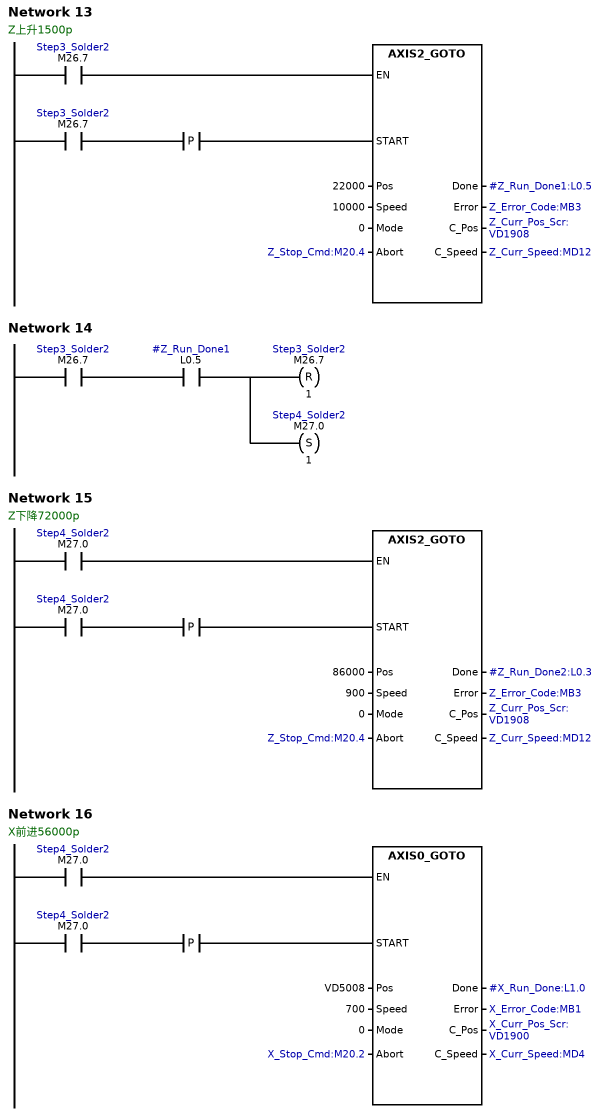
[picture p48: SBR39 networks 13-16]
Network 13
// Z上升1500p
LD     Step3_Solder2:M26.7
=      L60.0
LD     Step3_Solder2:M26.7
EU
=      L63.7
LD     L60.0
CALL   AXIS2_GOTO:SBR25, L63.7, 22000, 10000, 0, Z_Stop_Cmd:M20.4, #Z_Run_Done1:L0.5, Z_Error_Code:MB3, Z_Curr_Pos_Scr:VD1908, Z_Curr_Speed:MD12
Network 14
LD     Step3_Solder2:M26.7
A      #Z_Run_Done1:L0.5
R      Step3_Solder2:M26.7, 1
S      Step4_Solder2:M27.0, 1
Network 15
// Z下降72000p
LD     Step4_Solder2:M27.0
=      L60.0
LD     Step4_Solder2:M27.0
EU
=      L63.7
LD     L60.0
CALL   AXIS2_GOTO:SBR25, L63.7, 86000, 900, 0, Z_Stop_Cmd:M20.4, #Z_Run_Done2:L0.3, Z_Error_Code:MB3, Z_Curr_Pos_Scr:VD1908, Z_Curr_Speed:MD12
Network 16
// X前进56000p
LD     Step4_Solder2:M27.0
=      L60.0
LD     Step4_Solder2:M27.0
EU
=      L63.7
LD     L60.0
CALL   AXIS0_GOTO:SBR3, L63.7, VD5008, 700, 0, X_Stop_Cmd:M20.2, #X_Run_Done:L1.0, X_Error_Code:MB1, X_Curr_Pos_Scr:VD1900, X_Curr_Speed:MD4
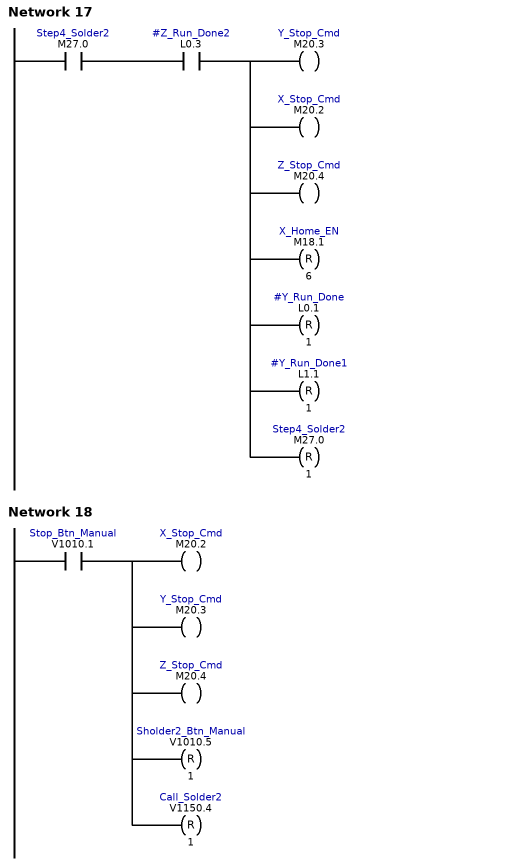
Network 17
LD     Step4_Solder2:M27.0
A      #Z_Run_Done2:L0.3
=      Y_Stop_Cmd:M20.3
=      X_Stop_Cmd:M20.2
=      Z_Stop_Cmd:M20.4
R      X_Home_EN:M18.1, 6
R      #Y_Run_Done:L0.1, 1
R      #Y_Run_Done1:L1.1, 1
R      Step4_Solder2:M27.0, 1
Network 18
LD     Stop_Btn_Manual:V1010.1
=      X_Stop_Cmd:M20.2
=      Y_Stop_Cmd:M20.3
=      Z_Stop_Cmd:M20.4
R      Sholder2_Btn_Manual:V1010.5, 1
R      Call_Solder2:V1150.4, 1
Network 23
// 程序段注释
END_SUBROUTINE_BLOCK

SUBROUTINE_BLOCK solder3:SBR40
TITLE=子例程注释
VAR_IN_OUT
Solder3_Cmd:BOOL;	// L0.0 
END_VAR
VAR
Y_Run_Done:BOOL;	// L0.1 
Z_Run_Done:BOOL;	// L0.2 
X_Run_Done:BOOL;	// L0.3 
Z_Run_Done2:BOOL;	// L0.4 
Z_Run_Done3:BOOL;	// L0.5 
Z_Run_Done4:BOOL;	// L0.6 
Z_Run_Done5:BOOL;	// L0.7 
Z_Run_Done6:BOOL;	// L1.0 
Z_Up_Done:BOOL;	// L1.1 
X_Run_Done2:BOOL;	// L1.2 
END_VAR
BEGIN
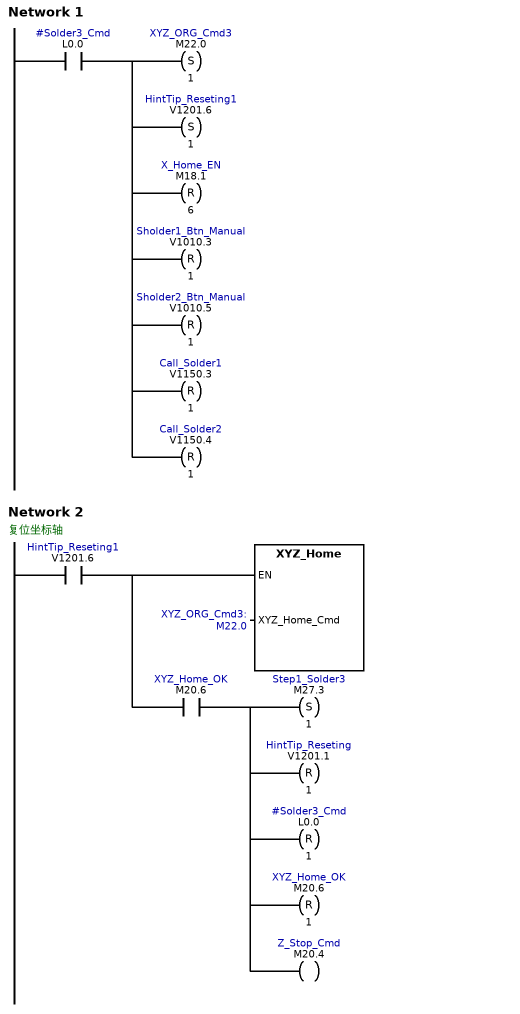
Network 1
LD     #Solder3_Cmd:L0.0
S      XYZ_ORG_Cmd3:M22.0, 1
S      HintTip_Reseting1:V1201.6, 1
R      X_Home_EN:M18.1, 6
R      Sholder1_Btn_Manual:V1010.3, 1
R      Sholder2_Btn_Manual:V1010.5, 1
R      Call_Solder1:V1150.3, 1
R      Call_Solder2:V1150.4, 1
Network 2
// 复位坐标轴
LD     HintTip_Reseting1:V1201.6
CALL   XYZ_Home:SBR37, XYZ_ORG_Cmd3:M22.0
A      XYZ_Home_OK:M20.6
S      Step1_Solder3:M27.3, 1
R      HintTip_Reseting:V1201.1, 1
R      #Solder3_Cmd:L0.0, 1
R      XYZ_Home_OK:M20.6, 1
=      Z_Stop_Cmd:M20.4
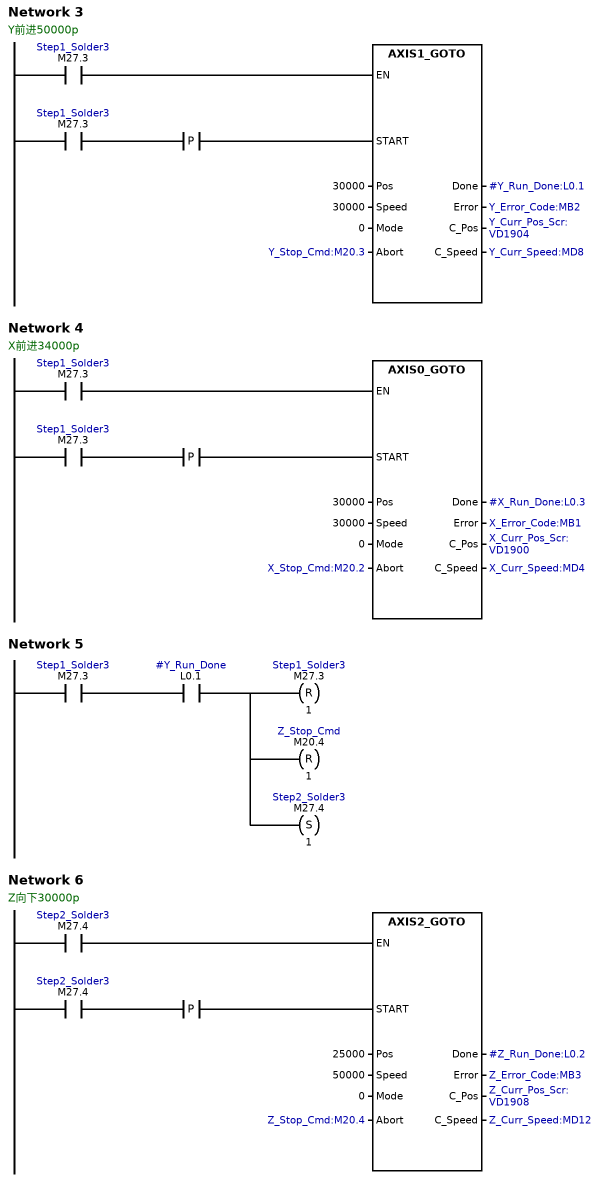
Network 3
// Y前进50000p
LD     Step1_Solder3:M27.3
=      L60.0
LD     Step1_Solder3:M27.3
EU
=      L63.7
LD     L60.0
CALL   AXIS1_GOTO:SBR14, L63.7, 30000, 30000, 0, Y_Stop_Cmd:M20.3, #Y_Run_Done:L0.1, Y_Error_Code:MB2, Y_Curr_Pos_Scr:VD1904, Y_Curr_Speed:MD8
Network 4
// X前进34000p
LD     Step1_Solder3:M27.3
=      L60.0
LD     Step1_Solder3:M27.3
EU
=      L63.7
LD     L60.0
CALL   AXIS0_GOTO:SBR3, L63.7, 30000, 30000, 0, X_Stop_Cmd:M20.2, #X_Run_Done:L0.3, X_Error_Code:MB1, X_Curr_Pos_Scr:VD1900, X_Curr_Speed:MD4
Network 5
LD     Step1_Solder3:M27.3
A      #Y_Run_Done:L0.1
R      Step1_Solder3:M27.3, 1
R      Z_Stop_Cmd:M20.4, 1
S      Step2_Solder3:M27.4, 1
Network 6
// Z向下30000p
LD     Step2_Solder3:M27.4
=      L60.0
LD     Step2_Solder3:M27.4
EU
=      L63.7
LD     L60.0
CALL   AXIS2_GOTO:SBR25, L63.7, 25000, 50000, 0, Z_Stop_Cmd:M20.4, #Z_Run_Done:L0.2, Z_Error_Code:MB3, Z_Curr_Pos_Scr:VD1908, Z_Curr_Speed:MD12
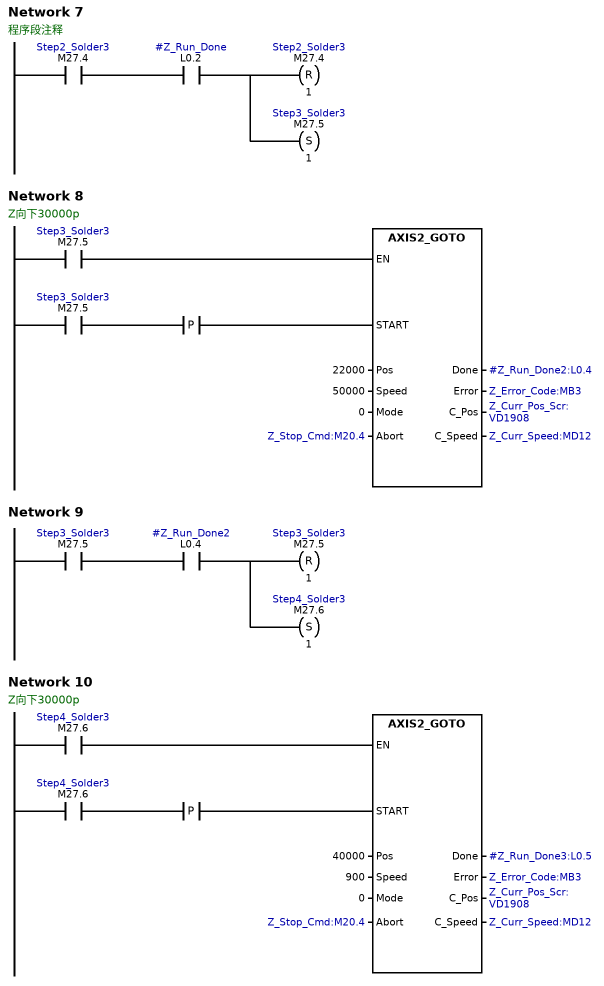
Network 7
// 程序段注释
LD     Step2_Solder3:M27.4
A      #Z_Run_Done:L0.2
R      Step2_Solder3:M27.4, 1
S      Step3_Solder3:M27.5, 1
Network 8
// Z向下30000p
LD     Step3_Solder3:M27.5
=      L60.0
LD     Step3_Solder3:M27.5
EU
=      L63.7
LD     L60.0
CALL   AXIS2_GOTO:SBR25, L63.7, 22000, 50000, 0, Z_Stop_Cmd:M20.4, #Z_Run_Done2:L0.4, Z_Error_Code:MB3, Z_Curr_Pos_Scr:VD1908, Z_Curr_Speed:MD12
Network 9
LD     Step3_Solder3:M27.5
A      #Z_Run_Done2:L0.4
R      Step3_Solder3:M27.5, 1
S      Step4_Solder3:M27.6, 1
Network 10
// Z向下30000p
LD     Step4_Solder3:M27.6
=      L60.0
LD     Step4_Solder3:M27.6
EU
=      L63.7
LD     L60.0
CALL   AXIS2_GOTO:SBR25, L63.7, 40000, 900, 0, Z_Stop_Cmd:M20.4, #Z_Run_Done3:L0.5, Z_Error_Code:MB3, Z_Curr_Pos_Scr:VD1908, Z_Curr_Speed:MD12
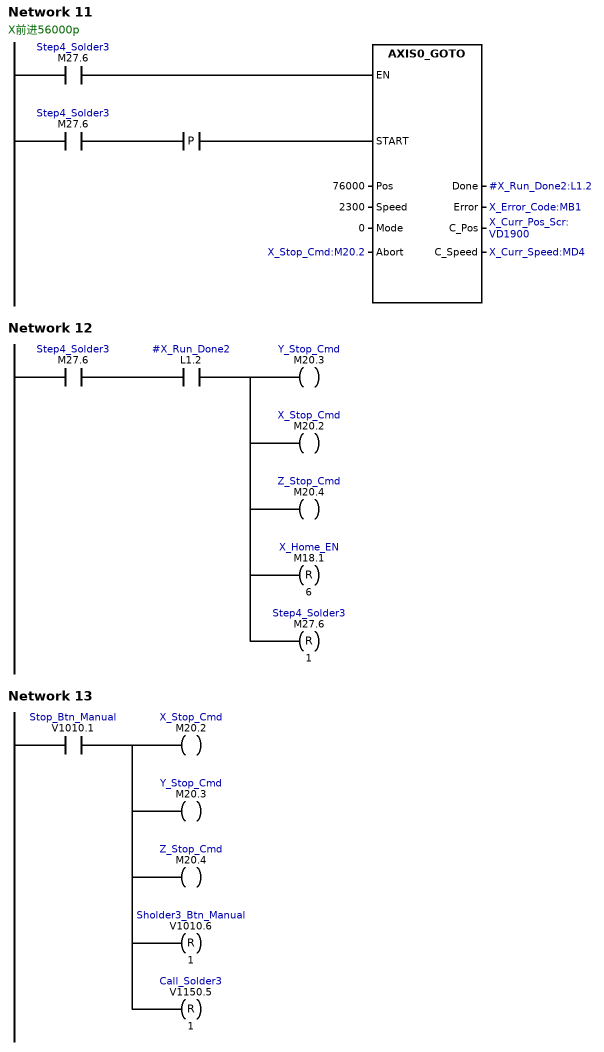
Network 11
// X前进56000p
LD     Step4_Solder3:M27.6
=      L60.0
LD     Step4_Solder3:M27.6
EU
=      L63.7
LD     L60.0
CALL   AXIS0_GOTO:SBR3, L63.7, 76000, 2300, 0, X_Stop_Cmd:M20.2, #X_Run_Done2:L1.2, X_Error_Code:MB1, X_Curr_Pos_Scr:VD1900, X_Curr_Speed:MD4
Network 12
LD     Step4_Solder3:M27.6
A      #X_Run_Done2:L1.2
=      Y_Stop_Cmd:M20.3
=      X_Stop_Cmd:M20.2
=      Z_Stop_Cmd:M20.4
R      X_Home_EN:M18.1, 6
R      Step4_Solder3:M27.6, 1
Network 13
LD     Stop_Btn_Manual:V1010.1
=      X_Stop_Cmd:M20.2
=      Y_Stop_Cmd:M20.3
=      Z_Stop_Cmd:M20.4
R      Sholder3_Btn_Manual:V1010.6, 1
R      Call_Solder3:V1150.5, 1
END_SUBROUTINE_BLOCK

SUBROUTINE_BLOCK SBR_41:SBR41
TITLE=子程序注释
BEGIN
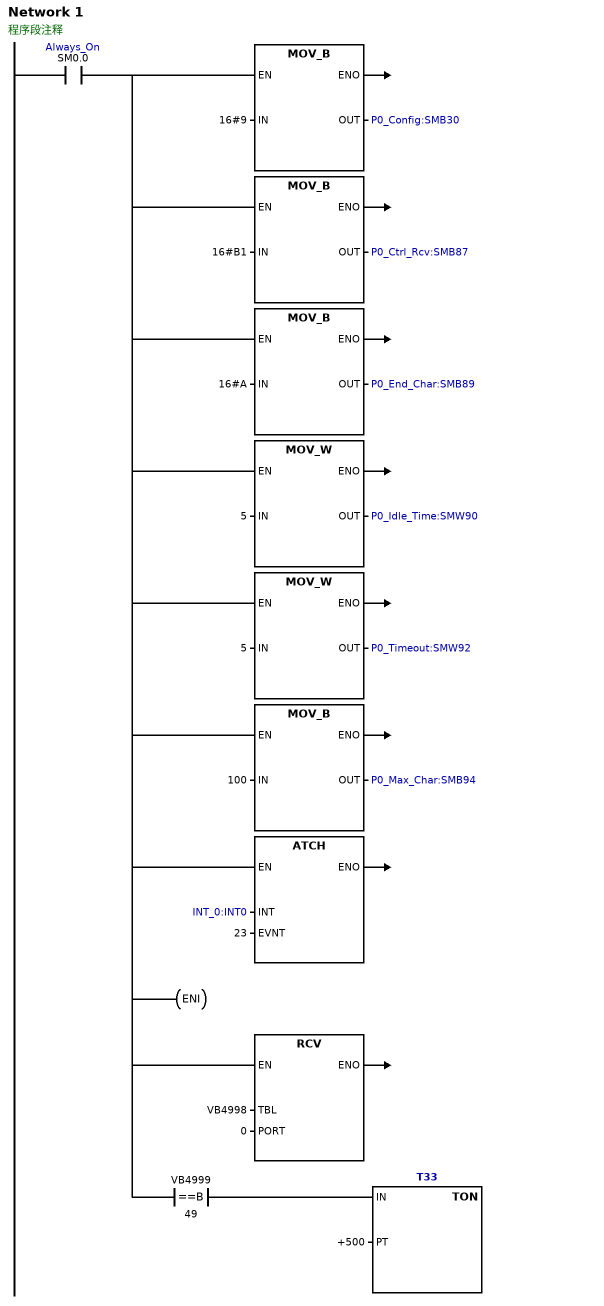
Network 1
// 程序段注释
LD     Always_On:SM0.0
MOVB   16#9, P0_Config:SMB30
MOVB   16#B1, P0_Ctrl_Rcv:SMB87
MOVB   16#A, P0_End_Char:SMB89
MOVW   5, P0_Idle_Time:SMW90
MOVW   5, P0_Timeout:SMW92
MOVB   100, P0_Max_Char:SMB94
ATCH   INT_0:INT0, 23
ENI
RCV    VB4998, 0
AB=    VB4999, 49
TON    T33, +500
Network 2
// 程序段注释
END_SUBROUTINE_BLOCK

INTERRUPT_BLOCK INT_0:INT0
TITLE=中断例程注释
BEGIN
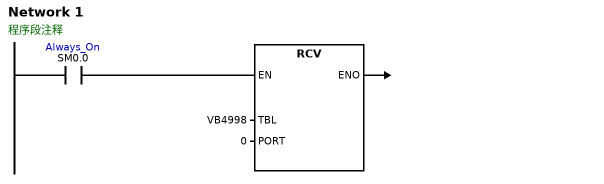
Network 1
// 程序段注释
LD     Always_On:SM0.0
RCV    VB4998, 0
END_INTERRUPT_BLOCK
